// TIA Portal V17 export
// export: Created 2025-08-05T09:35:59.1568817Z, ExportSetting WithDefaults, DisplayName Totally Integrated Automation Portal, DisplayVersion V17, DisplayName TIA Portal Openness, DisplayVersion V17, DisplayName TIA Portal Version Control Interface, DisplayVersion V17, DisplayName SINAMICS Startdrive Advanced, DisplayVersion V17, DisplayName SINAMICS Startdrive G130, G150, S120, S150, SINAMICS MV, S210, DisplayVersion V17, DisplayName SINAMICS Startdrive G110M, G120, G120C, G120D, G120P, G115D, DisplayVersion V17, DisplayName STEP 7 Professional, DisplayVersion V17, DisplayName STEP 7 Safety, DisplayVersion V17, DisplayName WinCC Advanced, DisplayVersion V17
VAR_GLOBAL   // PLC tag table "Default tag table"
   Start_Seq AT %M0.0 : Bool;
   Rob_Reset_1 AT %M0.1 : Bool;
   Rob_Reset_2 AT %M0.2 : Bool;
   RA_CC_1 AT %M0.3 : Bool;
END_VAR
VAR_GLOBAL CONSTANT   // user constants
   GRP_JOB_NAME_SIZE : Int := 50;   // String site group and job name / String Größe Gruppen- und Jobnamen
   MAX_CNT_GRP_OVR_ENTRIES : DInt := 100;   // Maximum number of groups in the group overview / Maximale Anzahl Gruppen in der Gruppen-Übersicht
   MAX_CNT_MTN_OVR_ENTRIES : DInt := 150;   // Maximum number of motions in the motion overview / Maximale Anzahl Motions in der Motion-Übersicht
END_VAR
